// TIA Portal project "风机燃气控制" (V17)

(* hardware
DEVICE "PLC_1"  S7-1200 Station
   slot 0: "Rack_0"  S7-1200 Rack  Rack  V1.0
   slot 1: "PLC_1"  CPU 1214C DC/DC/DC  6ES7 214-1AG40-0XB0  V4.5
*)

// ===== PLC "PLC_1"  CPU 1214C DC/DC/DC =====

VAR_GLOBAL   // PLC tag table "IO变量"
   "风机运行" AT %Q4.4 : Bool;
   "烧嘴电源" AT %Q4.6 : Bool;
   "风机控制" AT %QW44 : Word;
END_VAR

DATA_BLOCK "信号数据"   // DB1
{ S7_Optimized_Access := 'TRUE' }
VERSION : 0.1
   VAR
      风压测量值 : Real;   // 风压测量值(DBD80)
      风机手动 : Bool;   // 风机手动模式
      风机运行按 : Bool;   // 风机运行按钮
      风机自动输出 : Real;   // 风机自动输出值(DBD130)
      风机手动频率 : Real;   // 风机手动频率(DBD134)
      风机控制输出 : Real;   // 风机控制输出值(DBD138)
   END_VAR
BEGIN
END_DATA_BLOCK

DATA_BLOCK "内部数据"   // DB2
{ S7_Optimized_Access := 'TRUE' }
VERSION : 0.1
   VAR
      风压输出值 : Real;   // 风压转换计算输出
      风压过渡 : Int;   // 风压Real→Int过渡值
   END_VAR
BEGIN
END_DATA_BLOCK

DATA_BLOCK "数字量信号"   // DB3
{ S7_Optimized_Access := 'TRUE' }
VERSION : 0.1
   VAR
      风机故障反馈 : Bool;   // 风机故障反馈信号
   END_VAR
BEGIN
END_DATA_BLOCK

FUNCTION "风机燃气" : Void   // FC1, LAD
{ S7_Optimized_Access := 'TRUE' }
VERSION : 0.1
BEGIN

REGION Network 1
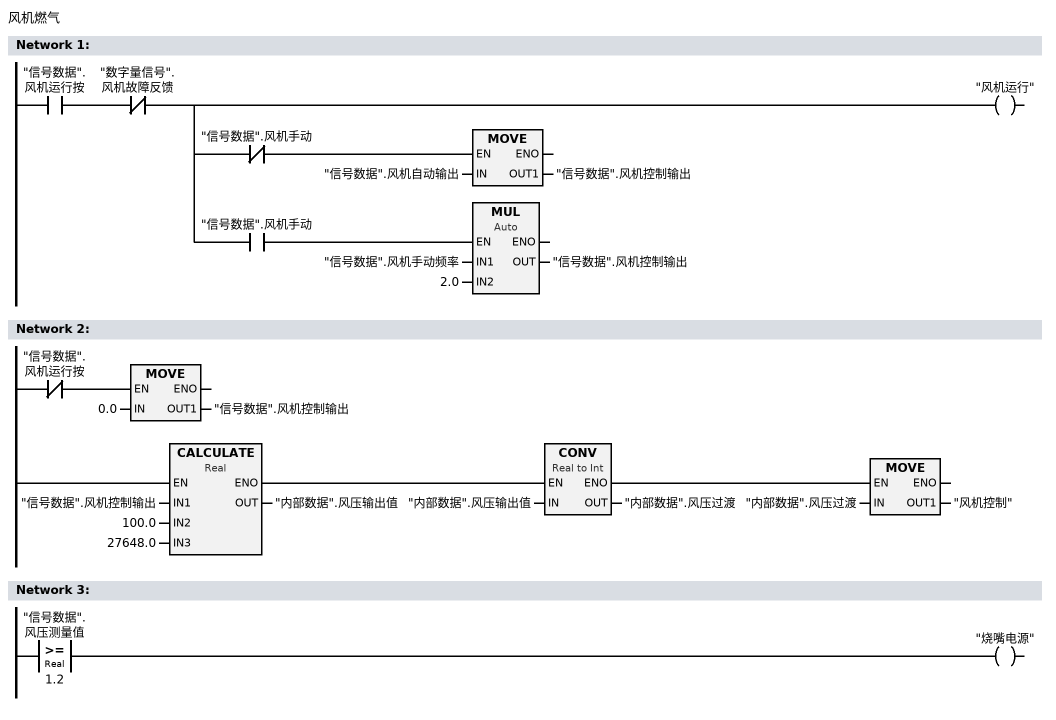
   RUNG wire#powerrail
      Contact( "信号数据".风机运行按 )
      I_Contact( "数字量信号".风机故障反馈 )
      wire#w1
      Coil( "风机运行" )
   END_RUNG
   RUNG wire#w1
      I_Contact( "信号数据".风机手动 )
      { S7_GenerateENO := "TRUE" } Move(in := "信号数据".风机自动输出, out1 => "信号数据".风机控制输出)
   END_RUNG
   RUNG wire#w1
      Contact( "信号数据".风机手动 )
      { S7_GenerateENO := "TRUE" } Mul(in1 := "信号数据".风机手动频率, in2 := 2.0, out => "信号数据".风机控制输出)
   END_RUNG
   // the same network as SCL:
   "风机运行" := "信号数据".风机运行按 AND NOT "数字量信号".风机故障反馈;
   IF "风机运行" AND NOT "信号数据".风机手动 THEN "信号数据".风机控制输出 := "信号数据".风机自动输出; END_IF;
   IF "风机运行" AND "信号数据".风机手动 THEN "信号数据".风机控制输出 := "信号数据".风机手动频率 * 2.0; END_IF;
END_REGION

REGION Network 2
   RUNG wire#powerrail
      I_Contact( "信号数据".风机运行按 )
      { S7_GenerateENO := "TRUE" } Move(in := 0.0, out1 => "信号数据".风机控制输出)
   END_RUNG
   RUNG wire#powerrail
      { S7_Templates := "SrcType := Real"; S7_GenerateENO := "TRUE"; S7_Expression := "(IN1/IN2)*IN3" } Calculate(in1 := "信号数据".风机控制输出, in2 := 100.0, in3 := 27648.0, out => "内部数据".风压输出值)
      { S7_Templates := "[SrcType := Real, DestType := Int]"; S7_GenerateENO := "TRUE" } Convert(in := "内部数据".风压输出值, out => "内部数据".风压过渡)
      { S7_GenerateENO := "TRUE" } Move(in := "内部数据".风压过渡, out1 => "风机控制")
   END_RUNG
   // the same network as SCL:
   // ENO of a box is taken as its EN; it also drops when the box reports an error
   IF NOT "信号数据".风机运行按 THEN "信号数据".风机控制输出 := 0.0; END_IF;
   "内部数据".风压输出值 := ("信号数据".风机控制输出/100.0)*27648.0;
   "内部数据".风压过渡 := REAL_TO_INT("内部数据".风压输出值);
   "风机控制" := "内部数据".风压过渡;
END_REGION

REGION Network 3
   RUNG wire#powerrail
      { S7_Templates := "SrcType := Real" } GE_Contact(in1 := "信号数据".风压测量值, in2 := 1.2)
      Coil( "烧嘴电源" )
   END_RUNG
   // the same network as SCL:
   "烧嘴电源" := "信号数据".风压测量值 >= 1.2;
END_REGION
END_FUNCTION

ORGANIZATION_BLOCK "Main"   // OB1, LAD, ProgramCycle
TITLE = "Main Program Sweep (Cycle)"
{ S7_Optimized_Access := 'TRUE' }
VERSION : 0.1
   VAR_INPUT
      Initial_Call : Bool;   // Initial call of this OB
      Remanence : Bool;   // =True, if remanent data are available
   END_VAR
BEGIN
END_ORGANIZATION_BLOCK